// TwinCAT 3 PLC project MyCustomLibraryPlcProject
// Title: My Custom Library
// Company: My Company
// Author: Your Name
// ProjectVersion: 1.2.3
// ProgramVersion: 3.1.4026.15
// libraries:
//   Tc2_System, * (Beckhoff Automation GmbH)
// project tree:
//   MyFunctions/ MyFunction.TcPOU

// ---- MyFunctions/MyFunction.TcPOU
FUNCTION MyFunction : T_MAXSTRING
VAR_INPUT
END_VAR
VAR
END_VAR

MyFunction := 'Hello World';

END_FUNCTION
